Staubli VAL3: toJointArrayRad.pgx

public program toJointArrayRad(jointRx& x_jJointRx, num& x_nJointArray[])
begin
  // Copyright (c) 2016, Ocado Technology - Robotics Research Team
  //
  // Licensed under the Apache License, Version 2.0 (the "License");
  // you may not use this file except in compliance with the License.
  // You may obtain a copy of the License at
  //
  //     http://www.apache.org/licenses/LICENSE-2.0
  //
  // Unless required by applicable law or agreed to in writing, software
  // distributed under the License is distributed on an "AS IS" BASIS,
  // WITHOUT WARRANTIES OR CONDITIONS OF ANY KIND, either express or implied.
  // See the License for the specific language governing permissions and
  // limitations under the License.

  // assuming the remaining elements (6-9) have zeros assigned by default
  x_nJointArray[0] = x_jJointRx.j1 * nDeg2Rad
  x_nJointArray[1] = x_jJointRx.j2 * nDeg2Rad
  x_nJointArray[2] = x_jJointRx.j3 * nDeg2Rad
  x_nJointArray[3] = x_jJointRx.j4 * nDeg2Rad
  x_nJointArray[4] = x_jJointRx.j5 * nDeg2Rad
  x_nJointArray[5] = x_jJointRx.j6 * nDeg2Rad
end
